FUNCTION_BLOCK "FB_EQP_PPI"
TITLE =%version: 0.06 % CN: 40
//Function:
//- Calculate displacement/plc scan
//- Make PPI one-shots on received PPI Pulse
//- Checking PPI error
//
//Description:
//On every leading or trailing edge from the PPI a one shot is generated
//On every PPI one shot the calculated displacement is corrected
//A PPI error is generated when a pulse is not seen within a sett time period.
//
//History:
//This version  %created_by: nlhdl %
//              %date_created: maandag 6 juli 2015 10:35:52 %
//              %release: VI_CONV/RA_Dev_Oakham %
//
//Modification History:                                   By:    Date:     Rev:
//----------------------------------------------------  -------  --------  -----
//7324: ECS-P General from the RD to RA for platform    nlHdL    06-07-15   0.06
//15807: Block consistency update IO symbols, comment   nlHdL    18-09-13   0.06
//CR19512 Update sources according S7 Manager           nlHdL    8-3-13   0.05
//CR19512 Update sources according S7 Manager           nlHdL    8-3-13   0.05
//PR8706 Preset error delay when no section run         nlHdL    09-01-12   0.04
//Minor changes for the major update                    nlMRe    16-09-10   0.03
//PR5145 PLT DB must have Done bit                      nlMRe    01-06-10   0.02
//Solved PR5102                                         nlMRe    16-04-10   0.01
//Renamed from FB_PPI
//
FAMILY : General
VERSION : 0.0


VAR_INPUT
  i_CFG_PPI_Resolution : INT ;	//CFG: [mm] Travel distance of belt, to generate 1 PPI-pulse (hardware setting)
  i_CFG_Time_Out_Error : INT ;	//CFG: [msec] Time before a PPI error is created
  i_DB_PLT : BLOCK_DB ;	//Data structure: Position datablock
  i_IO_PPI : BOOL ;	//HW: The PPI signal
  i_CMD_Reset : BOOL ;	//CMD: Reset command
END_VAR
VAR_OUTPUT
  o_PPI_Displacement_mm : INT ;	//The PPI displacement in [mm]
  o_ST_PPI_Err : BOOL ;	//ST: PPI Error
END_VAR
VAR
  s_Error_Delay : INT ;	//Timer PPI Error
  s_Copy_FP_PPI : BOOL ;	//Positive flank detection of PPI block-signal
  s_Copy_FN_PPI : BOOL ;	//Negative flank detection of PPI block-signal
  s_Section_Run : BOOL ;	//PLT: Section is running
  s_OS_PPI : BOOL ;	//One Shot of the PPI
END_VAR
BEGIN
NETWORK
TITLE =AA:  Read PLT DB
//The PLT is opened to get the section run signal.
      OPN   #i_DB_PLT; // Open PLT DB

      A     DBX   10.1; // Read Section Run Signal
      =     #s_Section_Run;
NETWORK
TITLE =BA: Make PPI one-shots
//If the PPI is used, the PPI block-wave signal 'i_PPI' will be converted to an
//One-Shot-signal 't_OS_PPI' by using the positive an negative flank of block
//signal.
//                                    ____      ____      ____      ____
//'i_PPI'   (bock-wave signal):  ____|    |____|    |____|    |____|    |___
//
//'t_OS_PPI' (One-Shot signal):  ____|____|____|____|____|____|____|____|___
      A     #i_IO_PPI; // IF
      FP    #s_Copy_FP_PPI; // Positive flank of an PPI-pulse..
      O(    ;
      A     #i_IO_PPI; // OR negative flank PPI-pulse..
      FN    #s_Copy_FN_PPI;
      )     ;
      =     #s_OS_PPI; // .. THEN generate PPI one-shot-pulses
NETWORK
TITLE =CA: Set/Reset PPI Error
//When the motor is running the error timer started. A new PPI pulse resets the
//timer with the default value. When the timer elaps a PPI error is set. The PPI
//error dissapears as soon as a reset is given.
      A     #i_CMD_Reset; //Reset PPI Error
      R     #o_ST_PPI_Err;

      A     #s_OS_PPI; //when a new pulse is seen
      O     #o_ST_PPI_Err; //..Or when there is a PPI error
      O     "M_First_Scan"; //..OR it is the first scan
      ON    #s_Section_Run; //..OR no section run
      JCN   CA01;

      L     #i_CFG_Time_Out_Error; //Set the default value in the timer.
      T     #s_Error_Delay;

CA01: A     #s_Section_Run; //If the section is running
      JCN   CA99;

      L     #s_Error_Delay; //Count down the PPI Error timer
      L     "MW_Prev_Cycle_Time";
      -I    ;
      JP    CA02; //If the error timer is below zero
      S     #o_ST_PPI_Err;
      L     0; //set back to zero
CA02: T     #s_Error_Delay; //Set new value in timer

CA99: NOP   0;
NETWORK
TITLE =DA: Calculate and write displacement
//If there is a PPI pulse, write the displacement in [mm] in the output.
      L     0; //Set current displacement output to zero.
      T     #o_PPI_Displacement_mm;

      A     #s_OS_PPI; //If there is a PPI pulse
      AN    #o_ST_PPI_Err; //..And no PPI error is active
      JCN   DA99;

      L     #i_CFG_PPI_Resolution; //Then write the current displacement (is same as resolution!)
      T     #o_PPI_Displacement_mm; //To the output.

DA99: NOP   0;
END_FUNCTION_BLOCK

